// TIA Portal V19 export
DATA_BLOCK "DB_ProductionRecords"   // DB76
{ S7_Optimized_Access := 'TRUE'; DB_Accessible_From_OPC_UA := 'FALSE' }
// stored: AutoNumber false, DBAccessibleFromOPCUA false, DBAccessibleFromWebserver false, MemoryReserve 100
   VAR RETAIN
      uiNumberOfRecords { ExternalWritable := 'False'} : UInt;
      aProdData { ExternalWritable := 'False'} : Array[0..200] of "stProductionRecord";
   END_VAR
BEGIN
END_DATA_BLOCK
